VAR_GLOBAL
	
	// 	Heartbeats from Stations OK
	gConsumed_Stn051ToSafetyInterface_OK : BOOL;
	gConsumed_Stn052ToSafetyInterface_OK : BOOL;
	gConsumed_Stn053ToSafetyInterface_OK : BOOL;
	gConsumed_Stn054ToSafetyInterface_OK : BOOL;	
	gConsumed_Stn055ToSafetyInterface_OK : BOOL;

	// PLC to PLC comms	
	gProduced_SafetyInterfaceConv : Plc2PlcDataSafetyPuckConv;
	gConsumed_Stn051ToSafetyInterface : Plc2PlcDataSafetyPuckConv;
	gConsumed_Stn052ToSafetyInterface : Plc2PlcDataSafetyPuckConv;
	gConsumed_Stn053ToSafetyInterface : Plc2PlcDataSafetyPuckConv;
	gConsumed_Stn054ToSafetyInterface : Plc2PlcDataSafetyPuckConv;
	gConsumed_Stn055ToSafetyInterface : Plc2PlcDataSafetyPuckConv;
	
	gInitialScanForce: BOOL := 0;
			
END_VAR

(* stored: Version 1.1.0.1, ProductVersion 3.1.4024.6
   GVL Global_Variables: Id {56202fa9-4423-49ed-a3ae-b1f78b12e440} *)
